// TIA Portal V17 export
// export: Created 2025-06-26T06:49:32.1912433Z, ExportSetting WithDefaults, DisplayName Totally Integrated Automation Portal, DisplayVersion V17 Update 8, DisplayName TIA Portal Openness, DisplayVersion V17 Update 8, DisplayName TIA Portal Version Control Interface, DisplayVersion V17, DisplayName STEP 7 Professional, DisplayVersion V17 Update 8, DisplayName STEP 7 Safety, DisplayVersion V17 Update 6, DisplayName WinCC Advanced, DisplayVersion V17 Update 8
TYPE "SystemData-STRUCT"
// stored: IsFailsafeCompliant false
   STRUCT
      SystemTypeNumber : Int;
      Limits : Struct
         T_SuperHeatCompressorIn_Min : Real;
         T_Housing_Max : Real;
         T_CoolingCycle_Max : Real;
         p_CompressorOut_Max : Real;
         p_EvaporatorOut_Max : Real;
      END_STRUCT;
      Constant : Bool;
      Settings : Struct
         CooliungPump_ReversedPWM : Bool;
         MotorCooling_AirFanCooledCycle : Bool;   // True if Air fan cooled otherwiese cooled via heat source cycle. Deactivates oil conditioning/prewarming
         DoubleExpansionValves : Bool;   // If A2 and B2 are present in the system
         Reserve3 : Bool;
         Reserve4 : Bool;
         Reserve5 : Bool;
      END_STRUCT;
   END_STRUCT;
END_TYPE
